FUNCTION F_Concat6_Large : LongString
VAR_IN_OUT CONSTANT
   sOne : LongString;
   sTwo : LongString;
   sThree : LongString;
   sFour : LongString;
   sFive : LongString;
   sSix : LongString;
END_VAR
VAR
   str : LongString;
END_VAR

str := F_Concat5_Large(sTwo, sThree, sFour, sFive, sSix);
F_Concat6_Large :=
   F_ConcatLarge(
      sOne,
      str
   );

END_FUNCTION

(* stored: Version 1.1.0.1, ProductVersion 3.1.4024.9
   POU F_Concat6_Large: Id {3877e970-03ef-4a02-a195-62ac08a0495d}, SpecialFunc None *)
